(* IEC 61131-3 sources: RL_MAR/experiments/comparison/llm4plc/results/deepseek-ai-DeepSeek-V3.2_20260506_104945/20260506_125018, 4 files *)

(* ---- generated_code_iteration_0.st ---- *)
START_ST
FUNCTION_BLOCK DoughMixerControl
VAR_INPUT
    IngredientsDetected : BOOL;
END_VAR
VAR_OUTPUT
    MixingInProgress : BOOL;
END_VAR
VAR
    state : INT;
    prevIngredientsDetected : BOOL;
    MixingTimeElapsed : TIME;
    MixingTimeLimit : TIME := T#5S;
END_VAR

(* State definitions *)
CONSTANT
    STATE_IDLE : INT := 0;
    STATE_MIXING : INT := 1;
END_CONSTANT

(* Main execution logic *)
CASE state OF
    STATE_IDLE:
        (* Output *)
        MixingInProgress := FALSE;
        (* Timer holds value - no increment in IDLE state *)
        (* Check for rising edge to start mixing *)
        IF (IngredientsDetected AND NOT prevIngredientsDetected) THEN
            (* Reset timer and transition to MIXING state *)
            MixingTimeElapsed := T#0S;
            state := STATE_MIXING;
        END_IF;

    STATE_MIXING:
        (* Output *)
        MixingInProgress := TRUE;
        (* Increment timer by 1 second per PLC cycle *)
        MixingTimeElapsed := MixingTimeElapsed + T#1S;
        (* Check transition conditions *)
        IF (MixingTimeElapsed >= MixingTimeLimit) OR (NOT IngredientsDetected) THEN
            state := STATE_IDLE;
        END_IF;
END_CASE;

(* Update edge detection variable for next cycle *)
prevIngredientsDetected := IngredientsDetected;

END_FUNCTION_BLOCK
END_ST

(* ---- generated_code_iteration_1.st ---- *)
START_REASON
The validation feedback indicates that the CODESYS compiler encountered an unexpected token 'CONSTANT'. In Structured Text for CODESYS, constants are typically declared using the `VAR CONSTANT` section within the variable declaration blocks, not with a standalone `CONSTANT` keyword. The original code used a `CONSTANT` block, which is not valid CODESYS syntax. This caused the compiler error. To fix this, I need to move the constant declarations into a `VAR CONSTANT` section inside the `VAR` block. Additionally, I should ensure proper variable declarations and maintain the function block structure as required.
END_REASON

START_ST
FUNCTION_BLOCK DoughMixerControl
VAR_INPUT
    IngredientsDetected : BOOL;
END_VAR
VAR_OUTPUT
    MixingInProgress : BOOL;
END_VAR
VAR
    state : INT;
    prevIngredientsDetected : BOOL;
    MixingTimeElapsed : TIME;
    MixingTimeLimit : TIME := T#5S;
    STATE_IDLE : INT := 0;
    STATE_MIXING : INT := 1;
END_VAR

(* Main execution logic *)
CASE state OF
    STATE_IDLE:
        (* Output *)
        MixingInProgress := FALSE;
        (* Timer holds value - no increment in IDLE state *)
        (* Check for rising edge to start mixing *)
        IF (IngredientsDetected AND NOT prevIngredientsDetected) THEN
            (* Reset timer and transition to MIXING state *)
            MixingTimeElapsed := T#0S;
            state := STATE_MIXING;
        END_IF;

    STATE_MIXING:
        (* Output *)
        MixingInProgress := TRUE;
        (* Increment timer by 1 second per PLC cycle *)
        MixingTimeElapsed := MixingTimeElapsed + T#1S;
        (* Check transition conditions *)
        IF (MixingTimeElapsed >= MixingTimeLimit) OR (NOT IngredientsDetected) THEN
            state := STATE_IDLE;
        END_IF;
END_CASE;

(* Update edge detection variable for next cycle *)
prevIngredientsDetected := IngredientsDetected;

END_FUNCTION_BLOCK
END_ST

(* ---- generated_code_iteration_2.st ---- *)
START_REASON
The CODESYS compiler error "CASE标号要求文字或符号整型常量" translates to "CASE label requires a literal or symbolic integer constant." This indicates that in the CASE statement, the labels (STATE_IDLE and STATE_MIXING) must be integer constants, but in the current code, they are variables declared in the VAR section. In CODESYS Structured Text, CASE labels must be compile-time constants, not runtime variables. To fix this, I should declare STATE_IDLE and STATE_MIXING as constants using VAR CONSTANT, ensuring they are true constants rather than mutable variables. Additionally, I'll move the MixingTimeLimit declaration to VAR CONSTANT as well since it's a fixed parameter. This will make the CASE statement valid and improve code clarity.
END_REASON

START_ST
FUNCTION_BLOCK DoughMixerControl
VAR_INPUT
    IngredientsDetected : BOOL;
END_VAR
VAR_OUTPUT
    MixingInProgress : BOOL;
END_VAR
VAR
    state : INT;
    prevIngredientsDetected : BOOL;
    MixingTimeElapsed : TIME;
END_VAR
VAR CONSTANT
    MixingTimeLimit : TIME := T#5S;
    STATE_IDLE : INT := 0;
    STATE_MIXING : INT := 1;
END_VAR

(* Main execution logic *)
CASE state OF
    STATE_IDLE:
        (* Output *)
        MixingInProgress := FALSE;
        (* Timer holds value - no increment in IDLE state *)
        (* Check for rising edge to start mixing *)
        IF (IngredientsDetected AND NOT prevIngredientsDetected) THEN
            (* Reset timer and transition to MIXING state *)
            MixingTimeElapsed := T#0S;
            state := STATE_MIXING;
        END_IF;

    STATE_MIXING:
        (* Output *)
        MixingInProgress := TRUE;
        (* Increment timer by 1 second per PLC cycle *)
        MixingTimeElapsed := MixingTimeElapsed + T#1S;
        (* Check transition conditions *)
        IF (MixingTimeElapsed >= MixingTimeLimit) OR (NOT IngredientsDetected) THEN
            state := STATE_IDLE;
        END_IF;
END_CASE;

(* Update edge detection variable for next cycle *)
prevIngredientsDetected := IngredientsDetected;

END_FUNCTION_BLOCK
END_ST

(* ---- generated_code_iteration_3.st ---- *)
START_REASON
The validation feedback indicates an encoding issue: "'gbk' codec can't decode byte 0xac in position 68: illegal multibyte sequence." This suggests that there might be a non-ASCII character (like a special quote or dash) in the code that's causing problems with the GBK encoding. Looking at the previous ST code, I notice that the comments contain standard ASCII characters, but there might be hidden or invisible non-ASCII characters introduced during copy-paste or formatting. To fix this, I'll ensure all characters in the code are plain ASCII by rewriting the comments and checking for any special symbols. Additionally, I'll maintain the FUNCTION_BLOCK structure with proper variable sections and CASE statement using constants. I'll also ensure the timer logic is correct by using a proper time increment method (though the current approach of adding T#1S per cycle is acceptable for simulation). The encoding error is likely due to a stray character, so I'll regenerate the code cleanly.
END_REASON

START_ST
FUNCTION_BLOCK DoughMixerControl
VAR_INPUT
    IngredientsDetected : BOOL;
END_VAR
VAR_OUTPUT
    MixingInProgress : BOOL;
END_VAR
VAR
    state : INT;
    prevIngredientsDetected : BOOL;
    MixingTimeElapsed : TIME;
END_VAR
VAR CONSTANT
    MixingTimeLimit : TIME := T#5S;
    STATE_IDLE : INT := 0;
    STATE_MIXING : INT := 1;
END_VAR

(* Main execution logic *)
CASE state OF
    STATE_IDLE:
        (* Output *)
        MixingInProgress := FALSE;
        (* Timer holds value - no increment in IDLE state *)
        (* Check for rising edge to start mixing *)
        IF (IngredientsDetected AND NOT prevIngredientsDetected) THEN
            (* Reset timer and transition to MIXING state *)
            MixingTimeElapsed := T#0S;
            state := STATE_MIXING;
        END_IF;

    STATE_MIXING:
        (* Output *)
        MixingInProgress := TRUE;
        (* Increment timer by 1 second per PLC cycle *)
        MixingTimeElapsed := MixingTimeElapsed + T#1S;
        (* Check transition conditions *)
        IF (MixingTimeElapsed >= MixingTimeLimit) OR (NOT IngredientsDetected) THEN
            state := STATE_IDLE;
        END_IF;
END_CASE;

(* Update edge detection variable for next cycle *)
prevIngredientsDetected := IngredientsDetected;

END_FUNCTION_BLOCK
END_ST
